ABB RobotStudio station: Brixey_6700.rsstn

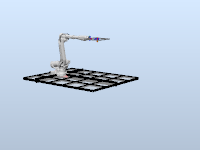
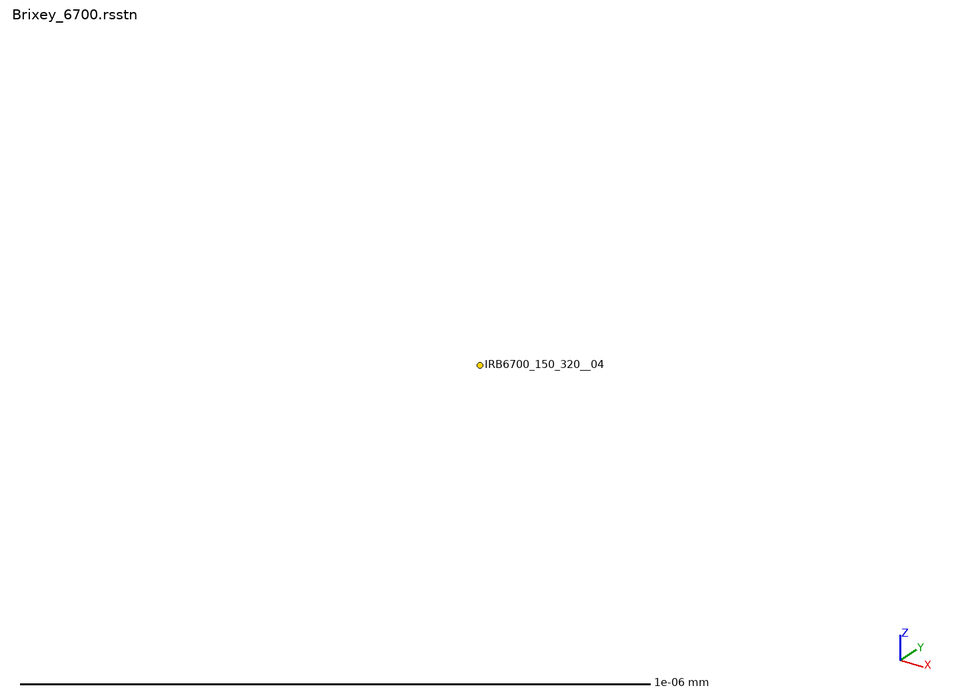
[picture v1: parts stored in the station drawn from their meshes, with robot base, taught points and paths (robot models come from the ABB library and are not in the file)]
Station Brixey_6700 (saved by RobotStudio 21.2.9526.0)
Controller IRB6700_150_320
  mechanical unit ROB_1: IRB6700_150_320__04, 6 joints, base frame (0, 0, 0) mm
Layout (positions relative to the parent item):
  - IRB6700_150_320__04 [mechanism, from Robots\IRB6700_150_320__04.rslib] at (0, 0, 0) mm; joint values [0.0237, -0.0221, 0.0301, 0, -0.008, 0] (rad or m)
  - plane [part] at (2582.43, 61.17, 2234.72) mm, rotated rx -180 ry -0.53 rz -178.64 deg, size 1000 x 1000 x 50 mm
  - Frame_1 [frame] at (2586.58, 0, 2203.66) mm
Attachment: plane is attached to IRB6700_150_320__04 / Link6
Targets, tools, work objects and paths stored in the station, written as RAPID:
! task T_ROB1
MODULE CalibData
  TASK PERS tooldata Tooldata_9:=[TRUE,[[43.288,0,500.872],[0.707106781,0,-0.707106781,0]],[1,[0,0,1],[1,0,0,0],0,0,0]];
  TASK PERS wobjdata Workobject_2:=[FALSE,TRUE,"",[[310.602096558,-31.145122511,792.988245486],[1,0,0,0]],[[0,0,0],[1,0,0,0]]];
ENDMODULE

